TYPE E_AteqProgramSeqStateFlags :
(
	FifoResetComplete,
	AutoZeroComplete,   
	ProgramSelectComplete,
	ProgramRunComplete,
	ReadLastResultComplete,
	ReadFIFOComplete,
	ResetDeviceDone
);
END_TYPE

(* stored: Version 1.1.0.1, ProductVersion 3.1.4024.15
   DUT E_AteqProgramSeqStateFlags: Id {31d3b071-ef6e-44f1-9157-16ac65450b8e} *)
